FUNCTION_BLOCK AxisPowerTestSuite
VAR
	StubAxis : AXIS_REF;
	TestAxisPower : AxisPower(StubAxis);
	ReRun: BOOL;
END_VAR

DoesAxisAcceptEnable_Test();
RejectEnableWhenEnabled_Test();
IF ReRun THEN
	TestSuite.ReRunTests();
	ReRun := FALSE;
END_IF

METHOD DoesAxisAcceptEnable_Test : BOOL
VAR_INST
	Expected : HRESULT;
	Actual	 : HRESULT;
END_VAR
IF TestSuite.Test(__POUNAME()).ExecuteTest() THEN
	Expected := s_OK;
	Actual := TestAxisPower.Enable();
	TestAxisPower.Disable();
	TestSuite.Test(__POUNAME()).AssertEqual(Expected, Actual);
END_IF
END_METHOD

METHOD RejectEnableWhenEnabled_Test : BOOL
VAR_INST
	Expected : HRESULT;
	Actual	 : HRESULT;
END_VAR
IF TestSuite.Test(__POUNAME()).ExecuteTest() THEN
	Expected := s_OK;
	TestAxisPower.Enable();
	Actual := TestAxisPower.Enable();
	TestAxisPower.Disable();
	TestSuite.Test(__POUNAME()).AssertEqual(Expected, Actual);
END_IF
END_METHOD

END_FUNCTION_BLOCK

(* stored: Version 1.1.0.1
   POU AxisPowerTestSuite: Id {ac2625ce-9cae-4674-bbac-7fb3863ceb8a}, SpecialFunc None
   Method DoesAxisAcceptEnable_Test: Id {fe79904b-ba9b-4299-9251-955ef4cd651f}
   Method RejectEnableWhenEnabled_Test: Id {3a8db93e-7de7-40e7-bc08-d2e3cb8c9735} *)
